// Mitsubishi GX Works2 project: RecipeMixer   PLC: FX3U/FX3UC

PROGRAM MAIN
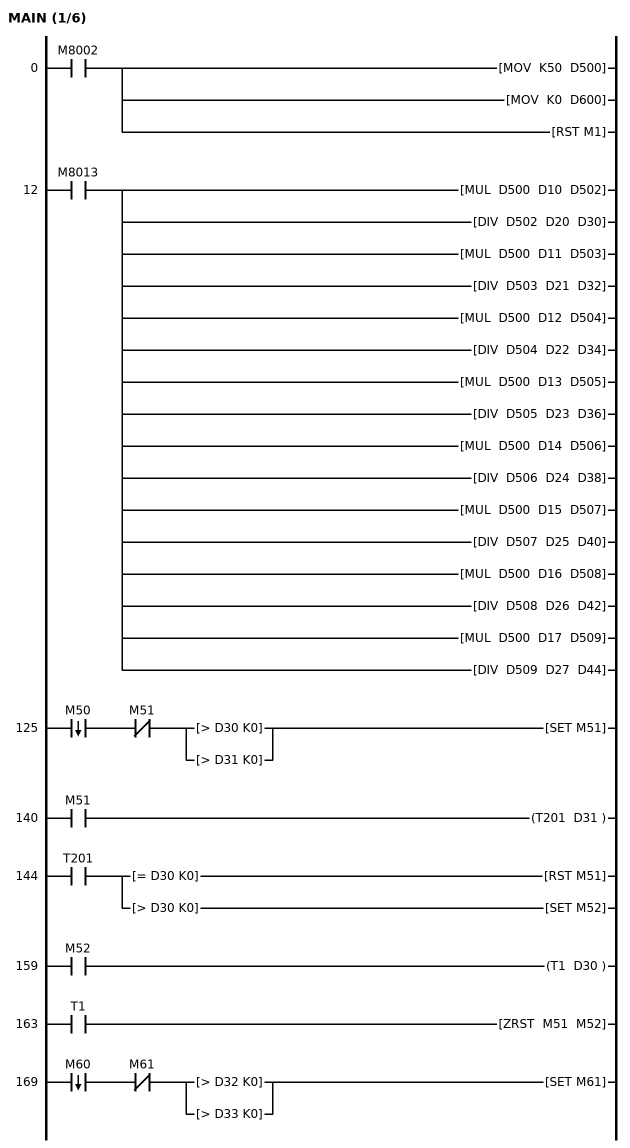
0     LD      M8002
      MOV     K50 D500
      MOV     K0 D600
      RST     M1
12    LD      M8013
      MUL     D500 D10 D502
      DIV     D502 D20 D30
      MUL     D500 D11 D503
      DIV     D503 D21 D32
      MUL     D500 D12 D504
      DIV     D504 D22 D34
      MUL     D500 D13 D505
      DIV     D505 D23 D36
      MUL     D500 D14 D506
      DIV     D506 D24 D38
      MUL     D500 D15 D507
      DIV     D507 D25 D40
      MUL     D500 D16 D508
      DIV     D508 D26 D42
      MUL     D500 D17 D509
      DIV     D509 D27 D44
125   LDF     M50
      ANI     M51
      LD>     D30 K0
      OR>     D31 K0
      ANB
      SET     M51
140   LD      M51
      OUT     T201 D31
144   LD      T201
      MPS
      AND=    D30 K0
      RST     M51
      MPP
      AND>    D30 K0
      SET     M52
159   LD      M52
      OUT     T1 D30
163   LD      T1
      ZRST    M51 M52
169   LDF     M60
      ANI     M61
      LD>     D32 K0
      OR>     D33 K0
      ANB
      SET     M61
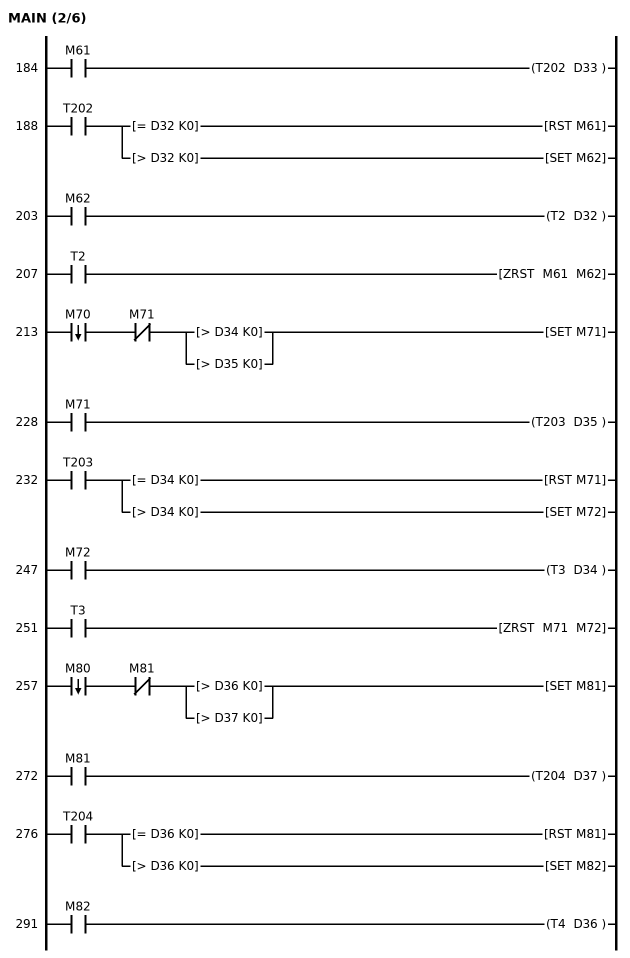
184   LD      M61
      OUT     T202 D33
188   LD      T202
      MPS
      AND=    D32 K0
      RST     M61
      MPP
      AND>    D32 K0
      SET     M62
203   LD      M62
      OUT     T2 D32
207   LD      T2
      ZRST    M61 M62
213   LDF     M70
      ANI     M71
      LD>     D34 K0
      OR>     D35 K0
      ANB
      SET     M71
228   LD      M71
      OUT     T203 D35
232   LD      T203
      MPS
      AND=    D34 K0
      RST     M71
      MPP
      AND>    D34 K0
      SET     M72
247   LD      M72
      OUT     T3 D34
251   LD      T3
      ZRST    M71 M72
257   LDF     M80
      ANI     M81
      LD>     D36 K0
      OR>     D37 K0
      ANB
      SET     M81
272   LD      M81
      OUT     T204 D37
276   LD      T204
      MPS
      AND=    D36 K0
      RST     M81
      MPP
      AND>    D36 K0
      SET     M82
291   LD      M82
      OUT     T4 D36
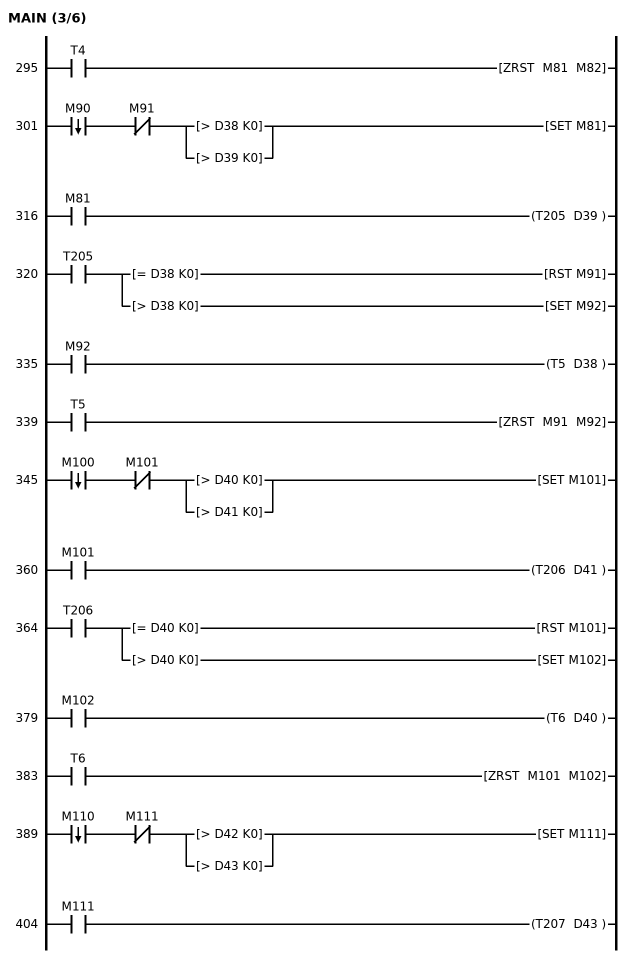
295   LD      T4
      ZRST    M81 M82
301   LDF     M90
      ANI     M91
      LD>     D38 K0
      OR>     D39 K0
      ANB
      SET     M81
316   LD      M81
      OUT     T205 D39
320   LD      T205
      MPS
      AND=    D38 K0
      RST     M91
      MPP
      AND>    D38 K0
      SET     M92
335   LD      M92
      OUT     T5 D38
339   LD      T5
      ZRST    M91 M92
345   LDF     M100
      ANI     M101
      LD>     D40 K0
      OR>     D41 K0
      ANB
      SET     M101
360   LD      M101
      OUT     T206 D41
364   LD      T206
      MPS
      AND=    D40 K0
      RST     M101
      MPP
      AND>    D40 K0
      SET     M102
379   LD      M102
      OUT     T6 D40
383   LD      T6
      ZRST    M101 M102
389   LDF     M110
      ANI     M111
      LD>     D42 K0
      OR>     D43 K0
      ANB
      SET     M111
404   LD      M111
      OUT     T207 D43
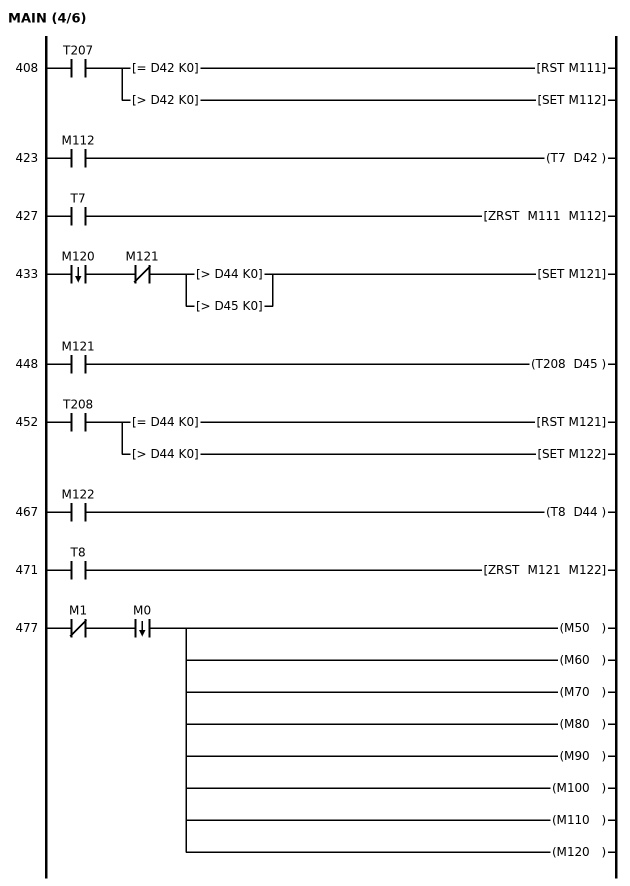
408   LD      T207
      MPS
      AND=    D42 K0
      RST     M111
      MPP
      AND>    D42 K0
      SET     M112
423   LD      M112
      OUT     T7 D42
427   LD      T7
      ZRST    M111 M112
433   LDF     M120
      ANI     M121
      LD>     D44 K0
      OR>     D45 K0
      ANB
      SET     M121
448   LD      M121
      OUT     T208 D45
452   LD      T208
      MPS
      AND=    D44 K0
      RST     M121
      MPP
      AND>    D44 K0
      SET     M122
467   LD      M122
      OUT     T8 D44
471   LD      T8
      ZRST    M121 M122
477   LDI     M1
      ANDF    M0
      OUT     M50
      OUT     M60
      OUT     M70
      OUT     M80
      OUT     M90
      OUT     M100
      OUT     M110
      OUT     M120
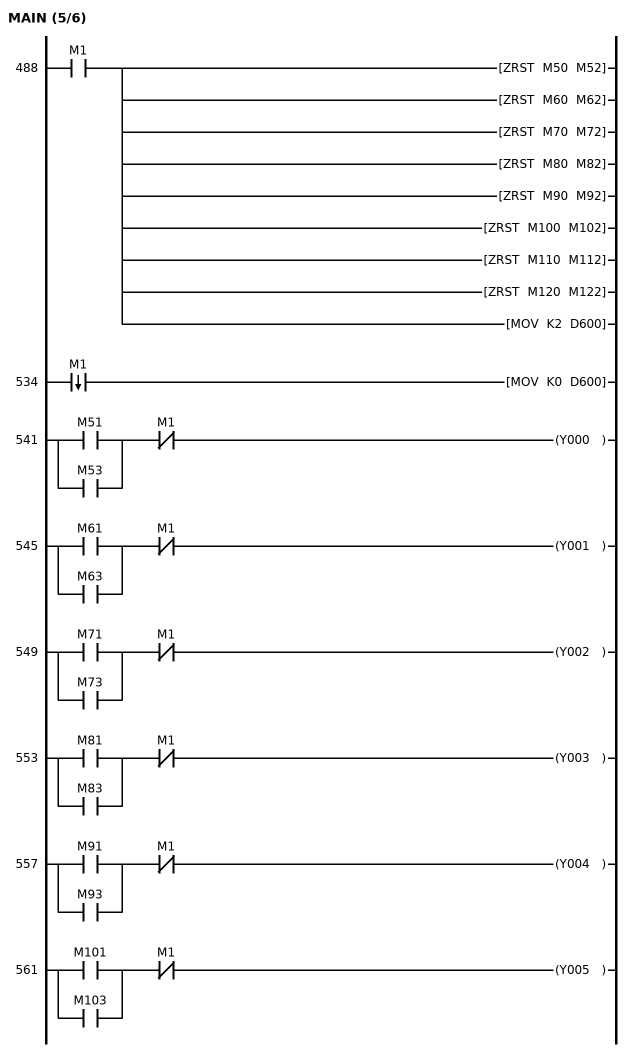
488   LD      M1
      ZRST    M50 M52
      ZRST    M60 M62
      ZRST    M70 M72
      ZRST    M80 M82
      ZRST    M90 M92
      ZRST    M100 M102
      ZRST    M110 M112
      ZRST    M120 M122
      MOV     K2 D600
534   LDF     M1
      MOV     K0 D600
541   LD      M51
      OR      M53
      ANI     M1
      OUT     Y000
545   LD      M61
      OR      M63
      ANI     M1
      OUT     Y001
549   LD      M71
      OR      M73
      ANI     M1
      OUT     Y002
553   LD      M81
      OR      M83
      ANI     M1
      OUT     Y003
557   LD      M91
      OR      M93
      ANI     M1
      OUT     Y004
561   LD      M101
      OR      M103
      ANI     M1
      OUT     Y005
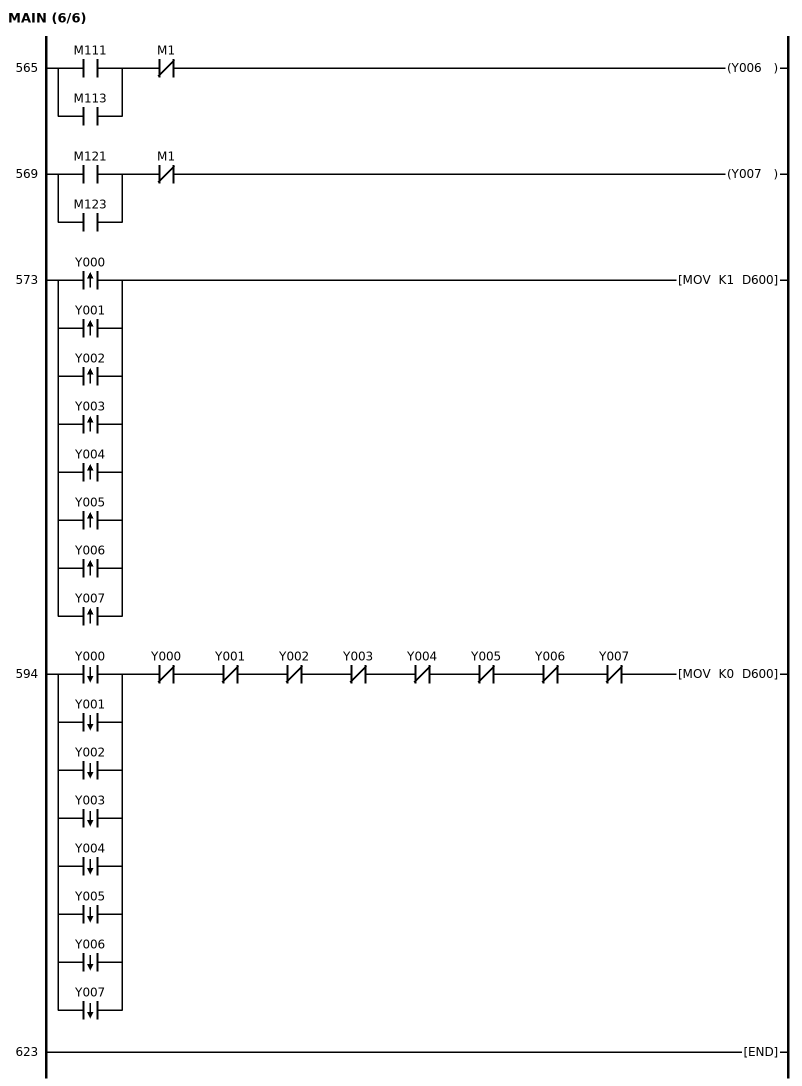
565   LD      M111
      OR      M113
      ANI     M1
      OUT     Y006
569   LD      M121
      OR      M123
      ANI     M1
      OUT     Y007
573   LDP     Y000
      ORP     Y001
      ORP     Y002
      ORP     Y003
      ORP     Y004
      ORP     Y005
      ORP     Y006
      ORP     Y007
      MOV     K1 D600
594   LDF     Y000
      ORF     Y001
      ORF     Y002
      ORF     Y003
      ORF     Y004
      ORF     Y005
      ORF     Y006
      ORF     Y007
      ANI     Y000
      ANI     Y001
      ANI     Y002
      ANI     Y003
      ANI     Y004
      ANI     Y005
      ANI     Y006
      ANI     Y007
      MOV     K0 D600
623   END
END_PROGRAM
